TYPE TcoCr800_Outputs_v_1_x_x :
STRUCT
	Outputs AT %Q* : ARRAY[0..63] OF BYTE;
END_STRUCT
END_TYPE

(* stored: Version 1.1.0.1, ProductVersion 3.1.4024.12
   DUT TcoCr800_Outputs_v_1_x_x: Id {3d53578d-1797-0756-06a2-1d6af208dec3} *)
